{attribute addProperty BoxType "AMP8000-0030-0103-0103"}
{attribute addProperty Id "FSoE_Master_CmdUSINT811Axis_A_STOBIT10.1251Safe_Output_1BIT10.1252Safe_Output_2BIT10.1253Safe_Output_3BIT10.1254Safe_Output_4BIT10.1255Safe_Output_5BIT10.1256Safe_Output_6BIT10.1257Safe_Output_7BIT10.1258Axis_B_STOBIT10.1259Safe_Output_9BIT10.12510Safe_Output_10BIT10.12511Safe_Output_11BIT10.12512Safe_Output_12BIT10.12513Safe_Output_13BIT10.12514Safe_Output_14BIT10.12515Safe_Output_15BIT10.12516FSoE_Master_CRC_0UINT1623FSoE_Master_ConnIDUINT1622"}
{attribute addProperty CRC "2786509782"}
{attribute addProperty SizeInBites "56"}
{attribute addProperty SizeInBytes "7"}
TYPE FSOE_A616C3D6 :
STRUCT
	{attribute addProperty Name "FSoE_Master_Cmd"}
	FSoE_Master_Cmd : USINT;
	{attribute addProperty Name "Axis_A_STO"}
	Axis_A_STO : BIT;
	{attribute addProperty Name "Safe_Output_1"}
	Safe_Output_1 : BIT;
	{attribute addProperty Name "Safe_Output_2"}
	Safe_Output_2 : BIT;
	{attribute addProperty Name "Safe_Output_3"}
	Safe_Output_3 : BIT;
	{attribute addProperty Name "Safe_Output_4"}
	Safe_Output_4 : BIT;
	{attribute addProperty Name "Safe_Output_5"}
	Safe_Output_5 : BIT;
	{attribute addProperty Name "Safe_Output_6"}
	Safe_Output_6 : BIT;
	{attribute addProperty Name "Safe_Output_7"}
	Safe_Output_7 : BIT;
	{attribute addProperty Name "Axis_B_STO"}
	Axis_B_STO : BIT;
	{attribute addProperty Name "Safe_Output_9"}
	Safe_Output_9 : BIT;
	{attribute addProperty Name "Safe_Output_10"}
	Safe_Output_10 : BIT;
	{attribute addProperty Name "Safe_Output_11"}
	Safe_Output_11 : BIT;
	{attribute addProperty Name "Safe_Output_12"}
	Safe_Output_12 : BIT;
	{attribute addProperty Name "Safe_Output_13"}
	Safe_Output_13 : BIT;
	{attribute addProperty Name "Safe_Output_14"}
	Safe_Output_14 : BIT;
	{attribute addProperty Name "Safe_Output_15"}
	Safe_Output_15 : BIT;
	{attribute addProperty Name "FSoE_Master_CRC_0"}
	FSoE_Master_CRC_0 : UINT;
	{attribute addProperty Name "FSoE_Master_ConnID"}
	FSoE_Master_ConnID : UINT;
END_STRUCT
END_TYPE

(* stored: Version 1.2.0.0, ProductVersion 3.1.4024.9
   DUT FSOE_A616C3D6: Id {8759b827-ef56-45f4-95a5-e68252dc4370} *)
